// TIA Portal V17 export
// export: Created 2022-07-20T06:59:39.5405894Z, ExportSetting WithDefaults, DisplayName Totally Integrated Automation Portal, DisplayVersion V17, DisplayName TIA Portal Openness, DisplayVersion V17, DisplayName TIA Portal Version Control Interface, DisplayVersion V17, DisplayName SINAMICS Startdrive Advanced, DisplayVersion V17, DisplayName SINAMICS Startdrive G130, G150, S120, S150, SINAMICS MV, S210, DisplayVersion V17, DisplayName SINAMICS Startdrive G110M, G120, G120C, G120D, G120P, G115D, DisplayVersion V17, DisplayName STEP 7 Professional, DisplayVersion V17, DisplayName STEP 7 Safety, DisplayVersion V17, DisplayName WinCC Advanced, DisplayVersion V17
FUNCTION "FC10015_IntToArray" : Void   // FC10015, LAD
TITLE = FC10015_IntToArray
{ S7_Optimized_Access := 'TRUE' }
AUTHOR : Jonathan
FAMILY : 1001x_CONVERT
VERSION : 1.0
// Release note : 
// 1.0 - Feature developped
// stored: AutoNumber false, IsIECCheckEnabled false, SetENOAutomatically false, UDAEnableTagReadback false
   VAR_INPUT
      Input_Int : Int;
   END_VAR
   VAR_OUTPUT
      Output_Array : Array[0..15] of Bool;
   END_VAR
   VAR_TEMP
      Temp_Word : Word;
   END_VAR
BEGIN

REGION Network 1 (SCL): Conversion Management
   #Temp_Word := INT_TO_WORD(#Input_Int);
   SCATTER(IN := #Temp_Word,
           OUT => #Output_Array);
END_REGION
END_FUNCTION
